// TIA Portal V19 export
DATA_BLOCK "LPythagorean_DB"   // DB3
// stored: InstanceOfName LPythagorean, InstanceOfType FB
"LPythagorean"
   // VAR_INPUT
   //    "a" : Int;
   //    "b" : Int;
   // END_VAR
   // VAR_OUTPUT
   //    c : Int;
   //    valid : Bool;
   // END_VAR
BEGIN
END_DATA_BLOCK
